Staubli VAL3: motionBuffer.pgx

public program motionBuffer(num x_nMovePts, num x_nElems)
begin

  // update motion buffer size

  userPageSet("uxMonitor", "lblMotionBuffer", "innerHTML", x_nElems)
  userPageSet("uxMonitor", "lblMotionBufferPopped", "innerHTML", x_nMovePts)

end
